ABB RAPID module: TCP_mtip_tool2.mod

MODULE TCP_mtip_tool2
	! Points are read in order of declaration.
  ! Please do not change the order of points!

  LOCAL PERS robtarget pTCP_Point1:=[[950.363,-124.222,476.374],[0.0596083365380764,-0.242846012115479,0.96697986125946,-0.0492195077240467],[-1,-3,1,1],[9E+09,9E+09,9E+09,9E+09,9E+09,9E+09]];
	LOCAL PERS robtarget pTCP_Point2:=[[875.3373,-428.1622,418.391],[0.168401315808296,-0.289312362670898,0.933462619781494,0.128790274262428],[-1,-2,0,1],[9E+09,9E+09,9E+09,9E+09,9E+09,9E+09]];
	LOCAL PERS robtarget pTCP_Point3:=[[1037.636,-433.0816,440.7565],[0.13380354642868,-0.713466048240662,0.679143369197845,0.108752444386482],[-1,-2,0,1],[9E+09,9E+09,9E+09,9E+09,9E+09,9E+09]];
	LOCAL PERS robtarget pTCP_Point4:=[[1106.607,-458.7698,430.0232],[0.132487788796425,-0.78712660074234,0.586081981658936,0.139235764741898],[-1,-2,0,1],[9E+09,9E+09,9E+09,9E+09,9E+09,9E+09]];
	LOCAL PERS robtarget pTCP_Point5:=[[970.7048,29.65234,452.1847],[0.0774419605731964,0.788783669471741,-0.595451056957245,0.1313816010952],[0,-3,1,1],[9E+09,9E+09,9E+09,9E+09,9E+09,9E+09]];
	LOCAL PERS robtarget pTCP_Point6:=[[1073.697,111.4896,429.5807],[0.0731830969452858,0.309505999088287,-0.930814027786255,0.180098548531532],[0,-3,2,1],[9E+09,9E+09,9E+09,9E+09,9E+09,9E+09]];

ENDMODULE
